FUNCTION_BLOCK PlcBasicNodePack IMPLEMENTS I_NodePack
VAR
	booleanLiteralNode : BooleanLiteralNode;
	booleanDisplayNode : BooleanDisplayNode;
END_VAR

METHOD PUBLIC RegisterWithNodeFactory
VAR_INPUT
	NodeFactory : I_NodeFactory;
END_VAR
NodeFactory.AddNodeAsPrototype('PlcBasic.Bool.BoolLiteral',booleanLiteralNode);
NodeFactory.AddNodeAsPrototype('PlcBasic.Bool.BoolDisplay',booleanDisplayNode);
END_METHOD

END_FUNCTION_BLOCK

(* stored: Version 1.1.0.1, ProductVersion 3.1.4024.12
   POU PlcBasicNodePack: Id {b1a7208c-fa6a-0ca2-104f-e5f6ddafa07d}, SpecialFunc None
   Method RegisterWithNodeFactory: Id {0a02d7c4-cf60-03c2-1373-451ec20f4e0e} *)
